INTERFACE I_CleaningStateCallback

METHOD mChangeState
VAR_INPUT
	sI_NextState : EN_Cleaning_State;
END_VAR
END_METHOD

METHOD mDeviceAbort : BOOL
VAR_INPUT
END_VAR
END_METHOD

METHOD mDeviceAckError
VAR_INPUT
END_VAR
END_METHOD

METHOD mDeviceOperation : BOOL
VAR_INPUT
	iI_Step : INT;	
END_VAR
END_METHOD

METHOD mSetMode : BOOL
VAR_INPUT
	sI_CleanMode	: EN_CLEANING_OP;
END_VAR
END_METHOD

PROPERTY pDeviceStatus : ST_CLEANING_DEV_STATUS
GET
END_GET
END_PROPERTY

END_INTERFACE

(* stored: Version 1.1.0.1, ProductVersion 3.1.4024.11
   Itf I_CleaningStateCallback: Id {9e2b1d7f-14a9-427c-91dc-aa99d83c1c41}
   Method mChangeState: Id {791fe484-0614-4ca3-8ffd-aa8144f1231d}
   Method mDeviceAbort: Id {f2c0cdde-162f-475f-807f-82c1b567a3c5}
   Method mDeviceAckError: Id {b3adda9e-4885-4832-8e5c-9cfffcdbe7e7}
   Method mDeviceOperation: Id {0860f684-1c2d-4ef9-9cb2-eb50cd1f317b}
   Method mSetMode: Id {17e00825-f735-4663-b79b-fcda0e4f1d96}
   Property pDeviceStatus: Id {f38ed1de-c880-4578-9def-59fb056d2d4b}
   Get Get: Id {9acb1614-cdf3-4ef8-b7e3-ba2f228e7879} *)
